PROGRAM ActuationSystems
VAR
fbMainJibCylinderHyd : ValveControlledCylinder;
//HydraulicCylinder
fbMainJibCylinderMech : CylinderMech;
fbHPU : HPU;
END_VAR

fbHPU(
);

//Hyd Model for MainJibCylinder
fbMainJibCylinderHyd(
	uDcvEnable := Inputs.uDcvEnableMainJib,
	uDcv := Inputs.uDcvMainJib,	
	ReturnPressure := G_ActuationSystems.ReturnPressure,
	SupplyPressure := G_ActuationSystems.SupplyPressure,
	par := Param.pMainJibCylinder,
	xPiston := fbMainJibCylinderMech.PistonPosition,
	vPiston := fbMainJibCylinderMech.PistonVelocity,
);

//Temp Mechanical Model for MainJibCylinder
fbMainJibCylinderMech(
	F_Hydraulic := fbMainJibCylinderHyd.F_Hydraulic,
	param := Param.pMainJibCylinder,
	F_Piston => Work.FpistonMainJib
);

END_PROGRAM

(* stored: Version 1.1.0.1, ProductVersion 3.1.4024.9
   POU ActuationSystems: Id {3cabdd9c-217f-443b-9923-404fabc5dbf5}, SpecialFunc None *)
